FUNCTION_BLOCK FB_PSp
VAR_INPUT
	Temp_Max: REAL;
	Temp_Min: REAL;

END_VAR
VAR_OUTPUT
	{attribute 'OPC.UA.DA' := '1'}Parameter	: ST_PSp_Parameter;		
	{attribute 'OPC.UA.DA' := '1'}Zustand		: ST_PSp_Zustand;	
END_VAR
VAR
	Zustandscheck		: FB_PSp_Zustandscheck;

	LeseDaten			: FB_PSp_Input;

	TF_oben			: FB_TF;
	TF_mitte		: FB_TF;
	TF_unten		: FB_TF;
END_VAR

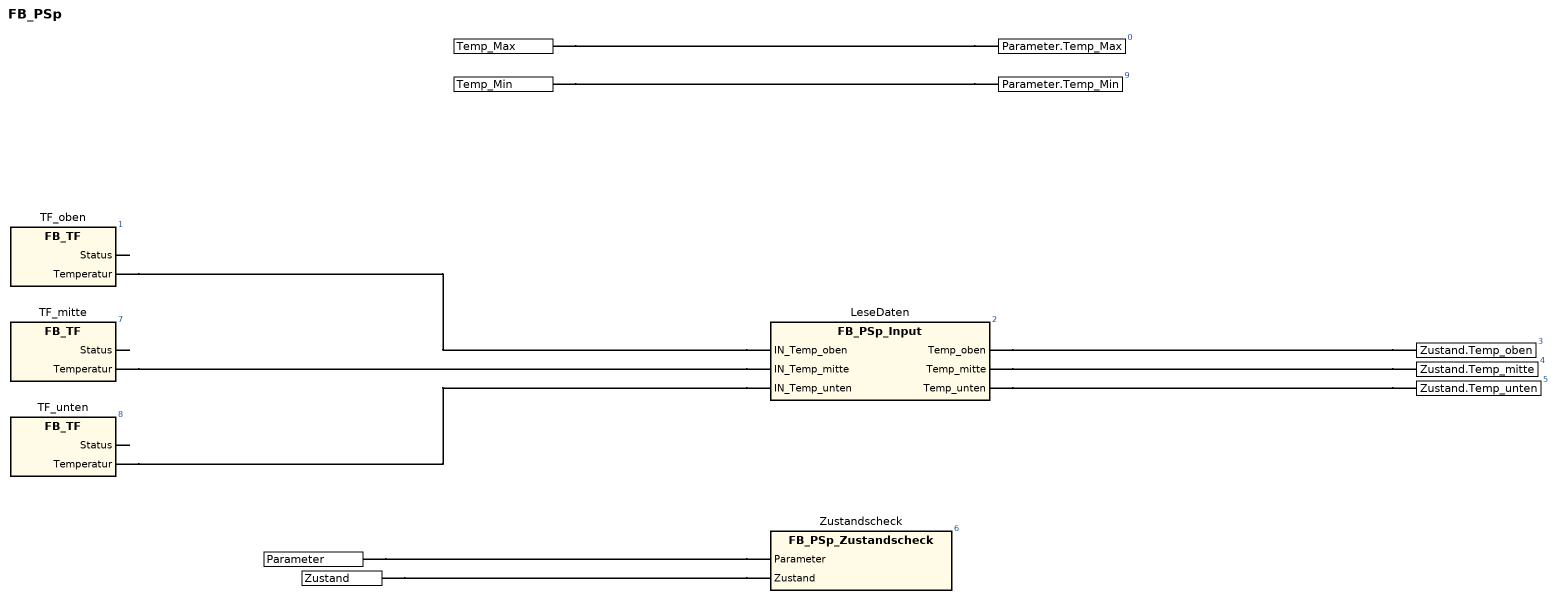
Parameter.Temp_Max := Temp_Max;
TF_oben(); // FB_TF
LeseDaten(
    IN_Temp_oben := TF_oben.Temperatur,
    IN_Temp_mitte := TF_mitte.Temperatur,
    IN_Temp_unten := TF_unten.Temperatur); // FB_PSp_Input
Zustand.Temp_oben := LeseDaten.Temp_oben;
Zustand.Temp_mitte := LeseDaten.Temp_mitte;
Zustand.Temp_unten := LeseDaten.Temp_unten;
Zustandscheck(Parameter := Parameter, Zustand := Zustand); // FB_PSp_Zustandscheck
TF_mitte(); // FB_TF
TF_unten(); // FB_TF
Parameter.Temp_Min := Temp_Min;

END_FUNCTION_BLOCK

(* stored: Version 1.1.0.1, ProductVersion 3.1.4024.9
   POU FB_PSp: Id {2c5d8db1-8ec1-472f-acd3-82a5106b438d}, SpecialFunc None *)
